{attribute 'GeneratedUsingTerminal: EPP1004-0061-0016'}
{attribute addProperty BoxType "EPP1004-0061-0016"}
{attribute addProperty Id "EtcSlaveTerminalBaseChannel_1AT %I*Channel_830843C11Channel_2AT %I*Channel_830843C11Channel_3AT %I*Channel_830843C11Channel_4AT %I*Channel_830843C11WcStateAT %I*WcState_9091E0EB2InfoDataAT %I*InfoData_6F19DB2B2"}
{attribute addProperty CRC "3213650938"}
{attribute addProperty Size "8"}
TYPE EPP1004_BF8C6BFA EXTENDS EtcSlaveTerminalBase :
STRUCT
	{attribute addProperty Name "Channel_1"}
	Channel_1 : Channel_830843C1;
	{attribute addProperty Name "Channel_2"}
	Channel_2 : Channel_830843C1;
	{attribute addProperty Name "Channel_3"}
	Channel_3 : Channel_830843C1;
	{attribute addProperty Name "Channel_4"}
	Channel_4 : Channel_830843C1;
	{attribute addProperty Name "WcState"}
	WcState : WcState_9091E0EB;
	{attribute addProperty Name "InfoData"}
	InfoData : InfoData_6F19DB2B;
END_STRUCT
END_TYPE

(* stored: Version 1.2.0.0, ProductVersion 3.1.4024.9
   DUT EPP1004_BF8C6BFA: Id {2931fedc-e8db-45db-86fd-e7efe3080782} *)
